PROGRAM P_Demo_MAXSTRING_TO_BYTEARR
VAR
    sTag    : STRING(255) := 'PumpAlpha-01'; // 工业语义：设备标签 STRING
    aBytes  : ARRAY[0..255] OF BYTE; // 字节数组输出
    bExport : BOOL; // 在线触发
END_VAR

// =============================================================================
// 场景：把配置文件中的 STRING 标签写入 ModBus 寄存器区（按字节数组对齐）。
// 价值：替代手写 FOR + 字节复制；本函数 1 调用。
// 验证步骤：
//   1. 引用 Tc2_Utilities
//   2. 编译 + 登录 + 运行
//   3. 在线写触发位 TRUE，monitor 输出变量
// =============================================================================

IF bExport THEN
    aBytes := MAXSTRING_TO_BYTEARR(in := sTag);
    bExport := FALSE;
END_IF;

END_PROGRAM

(* stored: Version 1.1.0.1, ProductVersion 3.1.4024.5
   POU P_Demo_MAXSTRING_TO_BYTEARR: Id {d14ecac8-a433-56ef-9804-5d7cf6a115d9}, SpecialFunc None *)
